{attribute 'GeneratedUsingTerminal: KL9900-0054'}
{attribute addProperty BoxType "KL9900-0054"}
{attribute addProperty Id "Channel_1AT %Q*Channel_60E28ED20"}
{attribute addProperty CRC "294106913"}
{attribute addProperty Size "0"}
TYPE KL_1187B721 :
STRUCT
	{attribute addProperty Name "Channel_1"}
	Channel_1 : Channel_60E28ED2;
END_STRUCT
END_TYPE

(* stored: Version 1.2.0.0, ProductVersion 3.1.4024.9
   DUT KL_1187B721: Id {51c44033-1d03-4d09-96c6-32ce288b61ab} *)
